FUNCTION_BLOCK FB_AxisHandautomatic
VAR_INPUT
    Notmoing:BOOL;//主轴停止中
	Run:BOOL;//自动
	i:INT;
	j: INT;
	Reset:BOOL;//手自动对比复位
END_VAR

VAR_OUTPUT
error :BOOL ;
END_VAR

VAR
	step:INT ;
	rRun : R_TRIG;
	fRun: F_TRIG;

	Pause_CMD:ARRAY[1..185] OF LREAL ; //手自动对比位置
	Handautomark:BOOL;//手自动对比标志
	K: INT;
	K1: INT;

END_VAR

VAR_IN_OUT

END_VAR




rRun(CLK:= Run , Q=> );
fRun(CLK:= Run , Q=> );


		IF fRun.Q THEN
			step:=100; 
		END_IF
		
	CASE step OF	
		100:
		   IF Notmoing THEN
			 step:=110;  
		   END_IF
	    110:    
	        Handautomark:=TRUE;
			FOR K:=i TO ((i+j)-1) DO 
			Pause_CMD[K]:=arrAxisCtrl[K].Status.fActPos;
			END_FOR
	        step:=120;    
	END_CASE
		

	   IF rRun.Q AND Handautomark THEN
				FOR K:=i TO ((i+j)-1) DO 
						IF  ABS(Pause_CMD[K]-arrAxisCtrl[K].Status.fActPos)>=0.2 THEN
						Axis_error[k]:=TRUE;
						END_IF
						
						IF Axis_error[k]   THEN
							error:=TRUE;
						END_IF
				END_FOR
				    Handautomark:=FALSE;
		END_IF
		
		IF stSysState.btnReset OR  stSysState.hmiReset  THEN
			   error:=FALSE;
			   FOR K1:=1 TO 185 DO 
				       Axis_error [K1]:=FALSE;
			   END_FOR
		END_IF
		
		IF Reset THEN
			 Handautomark:=FALSE;
		END_IF

END_FUNCTION_BLOCK

(* stored: Version 1.1.0.1, ProductVersion 3.1.4024.9
   POU FB_AxisHandautomatic: Id {56105043-b972-4bb8-8cec-3eeb00c73c96}, SpecialFunc None *)
